Staubli VAL3: load.pgx

public program load(string x_sItem, num& x_nResult)
  local string l_sType
  local string l_sPath
  local string l_sMessage
begin
  // load the select trajectory..already loaded
  call getTrajType(l_sType)
  if find(pt:libPath(),saveData:sPathTraj)==-1
    pt:libLoad(saveData:sPathTraj+l_sType)
    delay(0)
    if saveData:bDebug
      ? "loading HOME..."+saveData:sPathTraj+l_sType
    endIf
  endIf
  if isDefined(pt:tTraj[x_sItem])
    // use the type...
    call pt:link_it(x_sItem)
    jEditPoint=pt:tTraj[x_sItem]
    jEditPoint.sID=x_sItem
    x_nResult=0
  elseIf x_sItem!=""
    // not FOUND
    call language:message(l_sMessage,-7)
    x_nResult=-1
    popUpMsg(l_sMessage+x_sItem)
    jEditPoint.sID=""
  elseIf x_sItem==""
    // reload all the template
    call loadJoint("",x_nResult)
    call loadPoint("",x_nResult)
  endIf
end
